// TIA Portal V17 export
FUNCTION "MotorControl" : Void   // FC, LAD
{ S7_Optimized_Access := 'TRUE' }
VERSION : 0.1
// stored: AutoNumber true, IsIECCheckEnabled false, SetENOAutomatically false
BEGIN

REGION Network 1
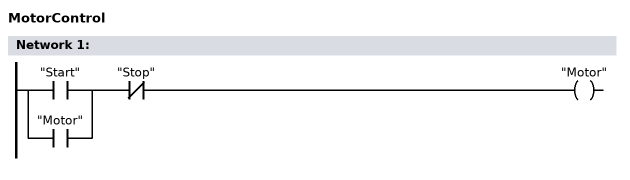
   RUNG wire#powerrail
      Contact( "Start" )
      wire#w1
      I_Contact( "Stop" )
      Coil( "Motor" )
   END_RUNG
   RUNG wire#powerrail
      Contact( "Motor" )
   END_RUNG wire#w1
   // the same network as SCL:
   "Motor" := ("Start" OR "Motor") AND NOT "Stop";
END_REGION
END_FUNCTION
